// TIA Portal V19 export
TYPE "C403_VAR_IF_SOS_TYPIC"
   STRUCT
      EXT_HW { ExternalAccessible := 'False'; ExternalVisible := 'False'; ExternalWritable := 'False'} : Bool;   // Sturings hardware (PLC) in storing
      STO { ExternalAccessible := 'False'; ExternalVisible := 'False'; ExternalWritable := 'False'} : Struct   // Opsomming van alle storingen
         A001 : Bool;   // Beveiliging aangesproken
         A002 : Bool;   // SOS-detectie is over 60 m tot 150 m uitgevallen
         A003 : Bool;   // SOS-detectie is over meer dan 150 m uitgevallen
      END_STRUCT;
   END_STRUCT;
END_TYPE
